// TIA Portal V18 export
// export: Created 2025-12-01T17:53:12.8409893Z, ExportSetting None, DisplayName Totally Integrated Automation Portal, DisplayVersion V18 Update 5, DisplayName TIA Portal Openness, DisplayVersion V18 Update 5, DisplayName TIA Portal Teamcenter Gateway, DisplayVersion V18, DisplayName TIA Portal Version Control Interface, DisplayVersion V18, DisplayName STEP 7 Professional, DisplayVersion V18 Update 5, DisplayName STEP 7 Safety, DisplayVersion V18, DisplayName WinCC Professional, DisplayVersion V18 Update 5
Screen "635 Analog Input"  1280x800, Number=635, Template=06Diagnosis
  ScreenLayer 
    TextField "文本域_2" at 75,185 size 76x32  StyleItem=TxtRight22, Text="××××"
    IOField "I/O 域_1" at 198,175 size 122x55  FormatPattern=s999.999, Mode=Output, StyleItem=I/O Display22
    Button "按钮_1" at 1024,725 size 128x75  StyleItem=BtnActive20, TextOff="模拟量 输入信号 / AI Input signal"
      on Click: ActivateScreen(Screen name := 616DP_Diagnosis, Object number := 0); SetTag(Tag := Sys_VersionManagement_HMIPageID, Value := 660)
    TextField "文本域_1" at 75,278 size 76x32  StyleItem=TxtRight22, Text="××××"
    IOField "I/O 域_2" at 198,268 size 122x55  FormatPattern=s999.999, Mode=Output, StyleItem=I/O Display22
      ProcessValue := 
    TextField "文本域_3" at 71,370 size 76x32  StyleItem=TxtRight22, Text="××××"
    IOField "I/O 域_3" at 198,361 size 122x55  FormatPattern=s999.999, Mode=Output, StyleItem=I/O Display22
      ProcessValue := 
    TextField "文本域_4" at 325,185 size 46x32  StyleItem=TxtRight22, Text="mm"
    TextField "文本域_5" at 323,278 size 20x32  StyleItem=TxtRight22, Text="N"
    TextField "文本域_6" at 324,371 size 40x32  StyleItem=TxtRight22, Text="bar"
